FUNCTION_BLOCK FB_ReadWrite_NC_PB
VAR_INPUT
	bReadParameter      : BOOL;
	bWriteParameter     : BOOL;
	iAxisNum            : INT;
	mcAxisParameter     : MC_AxisParameter;   //16#0001_0007 
END_VAR
VAR_OUTPUT
	fReadEncoderOffset  : LREAL;	
	bReatBusy           : BOOL;
	bWriteBusy          : BOOL;
	bReatError           : BOOL;
	bWriteError          : BOOL;
END_VAR
VAR
	mcReadParameter  : MC_ReadParameter;
	mcWriteParameter : MC_WriteParameter;	
END_VAR
VAR_IN_OUT
	fWriteEncoderOffset : LREAL;
END_VAR


mcReadParameter(
	Axis:= stAxis[iAxisNum] , 
	Enable:= bReadParameter , 
	ParameterNumber:= mcAxisParameter , 
	ReadMode:= , 
	Valid=> , 
	Busy=> bReatBusy , 
	Error=> bReatError , 
	ErrorID=> , 
	Value=>fReadEncoderOffset );
	
	
mcWriteParameter(
	Axis:= stAxis[iAxisNum] , 
	Execute:= bWriteParameter , 
	ParameterNumber:= mcAxisParameter, 
	Value:= fWriteEncoderOffset, 
	Done=> , 
	Busy=> bWriteBusy , 
	Error=> bWriteError , 
	ErrorID=> );

END_FUNCTION_BLOCK

(* stored: Version 1.1.0.1, ProductVersion 3.1.4024.11
   POU FB_ReadWrite_NC_PB: Id {d1e7d093-afc9-4066-85e9-84ac277ec7ec}, SpecialFunc None *)
